Staubli VAL3: DialogOnlyOK.pgx

public program dialogOnlyOK(string x_sTitle, string x_sText_r1, string x_sText_r2, string x_sText_r3, string x_sText_r4)
  local num l_nNum
begin

  //notes: screen size is 13rowsX40columns
  //usage: call DialogOnlyOK("RETURN IN HOME", "ATTENTION:", "Robot will return in home position", "be careful!", "", sUserScreen)

  wait(getKey()==-1)
  userPage()
  call clrscr()

  call sCenterTitle(x_sTitle)

  title(x_sTitle)

  gotoxy(0,4)
  call sCenterRow(x_sText_r1)
  putln(x_sText_r1)

  gotoxy(0,5)
  call sCenterRow(x_sText_r2)
  putln(x_sText_r2)

  gotoxy(0,6)
  call sCenterRow(x_sText_r3)
  putln(x_sText_r3)

  gotoxy(0,7)
  call sCenterRow(x_sText_r4)
  putln(x_sText_r4)

  gotoxy(0,13)
  put("F1=Ok")

  do
    l_nNum=get()
  until l_nNum==271

//  getKey()
//  while (getKey()!=271)
//    delay(0)
//  endWhile

  call clrscr()
  wait(getKey()==-1)

end
